PROGRAM MAIN
VAR
	
END_VAR

Habilita_Eixo();

END_PROGRAM

(* stored: Version 1.1.0.1
   POU MAIN: Id {df7afbcc-06d8-4e1b-9af1-bd4138249003}, SpecialFunc None *)
